TYPE BitStructure :
STRUCT
	Bit1 : BIT;
	Bit2 : BIT;
	Bit3 : BIT;
	Bit4 : BIT;
	Bit5 : BIT;
	Bit6 : BIT;
	Bit7 : BIT;
	Bit8 : BIT;	
END_STRUCT
END_TYPE

(* stored: Version 1.1.0.1, ProductVersion 3.1.4024.11
   DUT BitStructure: Id {4f93823c-2425-414d-8671-5350fceba74f} *)
